// TIA Portal project "AutomationProjectLMF" (V16)

(* hardware
DEVICE "S7-1200 station_1"  S7-1200 Station
   slot 0: "Telaio di montaggio_0"  S7-1200 Rack  Rack  V1.0
   slot 1: "PLC_1"  CPU 1215C AC/DC/Rly  6ES7 215-1BG40-0XB0  V4.2
*)

// ===== PLC "PLC_1"  CPU 1215C AC/DC/Rly =====

VAR_GLOBAL   // PLC tag table "Tabella delle variabili standard"
   "ARM_UP" AT %Q0.5 : Bool;
   "ARM_DOWN" AT %Q0.4 : Bool;
   "ArmTopStop" AT %I0.4 : Bool;
   "ARM_FRONT" AT %Q0.2 : Bool;
   "ARM_BACK" AT %Q0.3 : Bool;
   "FullBackArm" AT %I0.2 : Bool;
   "ARM_CCLOCKWISE" AT %Q0.7 : Bool;
   "ARM_CLOCKWISE" AT %Q0.6 : Bool;
   "FullyClockwiseArm" AT %I0.5 : Bool;
   "GRIP_CLOSE" AT %Q0.1 : Bool;
   "GRIP_OPEN" AT %Q0.0 : Bool;
   "FullyOpenGripper" AT %I0.0 : Bool;
   "RotationalEncoder" AT %ID1000 : DInt;
   "RotationalCounter" AT %MW2 : UInt;
   "VerticalEncoder" AT %ID1004 : DInt;
   "VerticalCounter" AT %MW4 : UInt;
   "System_Byte" AT %MB1 : Byte;
   "FirstScan" AT %M1.0 : Bool;
   "DiagStatusUpdate" AT %M1.1 : Bool;
   "AlwaysTRUE" AT %M1.2 : Bool;
   "AlwaysFALSE" AT %M1.3 : Bool;
   "System_Byte(1)" AT %MB1 : Byte;
   "System_Byte(2)" AT %MB1 : Byte;
   "System_Byte(3)" AT %MB1 : Byte;
   "Clock_Byte" AT %MB0 : Byte;
   "Clock_10Hz" AT %M0.0 : Bool;
   "Clock_5Hz" AT %M0.1 : Bool;
   "Clock_2.5Hz" AT %M0.2 : Bool;
   "Clock_2Hz" AT %M0.3 : Bool;
   "Clock_1.25Hz" AT %M0.4 : Bool;
   "Clock_1Hz" AT %M0.5 : Bool;
   "Clock_0.625Hz" AT %M0.6 : Bool;
   "Clock_0.5Hz" AT %M0.7 : Bool;
   "ForceReset" AT %M7.0 : Bool;
   "ResetCompleted" AT %M7.1 : Bool;
   "FRONT_STOP" AT %M7.2 : Bool;
   "ArmHCounter" AT %I0.3 : Bool;
   "ObjectDetected" AT %I1.5 : Bool;
   "HTarget" AT %MB2 : Byte;
   "Stop" AT %M6.1 : Bool;
   "GripperCounter" AT %I0.1 : Bool;
   "Started" AT %M6.3 : Bool;
   "FirstTarget" AT %M6.4 : Bool;
   "SecondTarget" AT %M6.5 : Bool;
   "ThirdTarget" AT %M6.6 : Bool;
   "Reset" AT %M6.7 : Bool;
   "FourthTarget" AT %M7.3 : Bool;
   "FifthTarget" AT %M7.4 : Bool;
   "SixthTarget" AT %M7.5 : Bool;
   "Conveyor" AT %Q1.1 : Bool;
   "Cart_Command" AT %MB3 : Byte;
   "Receveid_values" AT %MB4 : Byte;
   "CartReady" AT %M8.0 : Bool;
END_VAR

DATA_BLOCK "TCP_msg"   // DB8
{ S7_Optimized_Access := 'TRUE' }
VERSION : 0.1
   VAR
      Send : Byte := 0;
      Receive : Byte;
   END_VAR
BEGIN
END_DATA_BLOCK

// folder: System blocks/Program resources

DATA_BLOCK "ArmHPulseCounter"   // DB1
{ S7_Optimized_Access := 'TRUE' }
AUTHOR : Simatic
FAMILY : IEC
NAME : CNTR
VERSION : 1.0
// stored: InstanceOfName IEC_COUNTER
"IEC_COUNTER"
BEGIN
END_DATA_BLOCK

DATA_BLOCK "GripperPulseCounter"   // DB2
{ S7_Optimized_Access := 'TRUE' }
AUTHOR : Simatic
FAMILY : IEC
NAME : CNTR
VERSION : 1.0
// stored: InstanceOfName IEC_COUNTER
"IEC_COUNTER"
BEGIN
END_DATA_BLOCK

DATA_BLOCK "PLC_1_Connection_DB"   // DB5
{ S7_Optimized_Access := 'TRUE' }
AUTHOR : SIMATIC
FAMILY : MC7Plus
NAME : TC_IP_v4
VERSION : 1.0
// stored: InstanceOfName TCON_IP_v4
"TCON_IP_v4"
BEGIN
   ID := 1;
   InterfaceId := 64;
   RemotePort := 2001;
   ActiveEstablished := true;
   RemoteAddress.ADDR[1] := 192;
   RemoteAddress.ADDR[2] := 168;
   RemoteAddress.ADDR[4] := 241;
END_DATA_BLOCK

// folder: (top level)

ORGANIZATION_BLOCK "Main"   // OB1, LAD, ProgramCycle
TITLE = "Main Program Sweep (Cycle)"
{ S7_Optimized_Access := 'TRUE' }
VERSION : 0.1
   VAR_INPUT
      Initial_Call : Bool;   // Initial call of this OB
      Remanence : Bool;   // =True, if remanent data are available
   END_VAR
   VAR_TEMP   // added for the SCL form of the ladder/FBD networks
      _w1 : Bool;
      _w2 : Bool;
      _w3 : Bool;
   END_VAR
BEGIN

REGION Network 1
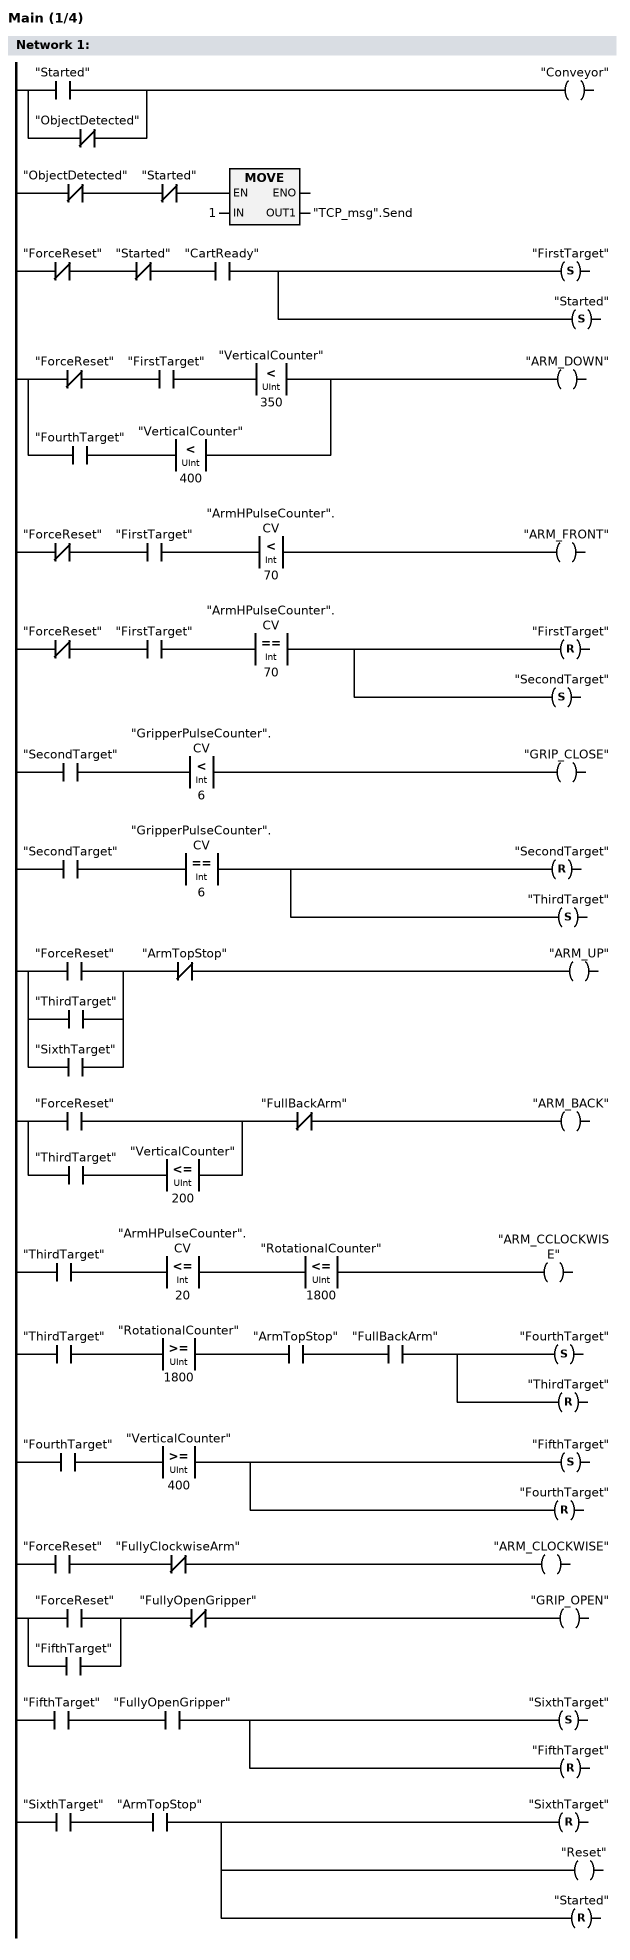
   RUNG wire#powerrail
      Contact( "Started" )
      wire#w1
      Coil( "Conveyor" )
   END_RUNG
   RUNG wire#powerrail
      I_Contact( "ObjectDetected" )
   END_RUNG wire#w1
   RUNG wire#powerrail
      I_Contact( "ObjectDetected" )
      I_Contact( "Started" )
      Move(in := 1, out1 => "TCP_msg".Send)
   END_RUNG
   RUNG wire#powerrail
      I_Contact( "ForceReset" )
      I_Contact( "Started" )
      Contact( "CartReady" )
      wire#w2
      S_Coil( "FirstTarget" )
   END_RUNG
   RUNG wire#w2
      S_Coil( "Started" )
   END_RUNG
   RUNG wire#powerrail
      I_Contact( "ForceReset" )
      Contact( "FirstTarget" )
      { S7_Templates := "SrcType := UInt" } LT_Contact(in1 := "VerticalCounter", in2 := 350)
      wire#w3
      Coil( "ARM_DOWN" )
   END_RUNG
   RUNG wire#powerrail
      Contact( "FourthTarget" )
      { S7_Templates := "SrcType := UInt" } LT_Contact(in1 := "VerticalCounter", in2 := 400)
   END_RUNG wire#w3
   RUNG wire#powerrail
      I_Contact( "ForceReset" )
      Contact( "FirstTarget" )
      { S7_Templates := "SrcType := Int" } LT_Contact(in1 := "ArmHPulseCounter".CV, in2 := 70)
      Coil( "ARM_FRONT" )
   END_RUNG
   RUNG wire#powerrail
      I_Contact( "ForceReset" )
      Contact( "FirstTarget" )
      { S7_Templates := "SrcType := Int" } EQ_Contact(in1 := "ArmHPulseCounter".CV, in2 := 70)
      wire#w4
      R_Coil( "FirstTarget" )
   END_RUNG
   RUNG wire#w4
      S_Coil( "SecondTarget" )
   END_RUNG
   RUNG wire#powerrail
      Contact( "SecondTarget" )
      { S7_Templates := "SrcType := Int" } LT_Contact(in1 := "GripperPulseCounter".CV, in2 := 6)
      Coil( "GRIP_CLOSE" )
   END_RUNG
   RUNG wire#powerrail
      Contact( "SecondTarget" )
      { S7_Templates := "SrcType := Int" } EQ_Contact(in1 := "GripperPulseCounter".CV, in2 := 6)
      wire#w5
      R_Coil( "SecondTarget" )
   END_RUNG
   RUNG wire#w5
      S_Coil( "ThirdTarget" )
   END_RUNG
   RUNG wire#powerrail
      Contact( "ForceReset" )
      wire#w6
      I_Contact( "ArmTopStop" )
      Coil( "ARM_UP" )
   END_RUNG
   RUNG wire#powerrail
      Contact( "ThirdTarget" )
   END_RUNG wire#w6
   RUNG wire#powerrail
      Contact( "SixthTarget" )
   END_RUNG wire#w6
   RUNG wire#powerrail
      Contact( "ForceReset" )
      wire#w7
      I_Contact( "FullBackArm" )
      Coil( "ARM_BACK" )
   END_RUNG
   RUNG wire#powerrail
      Contact( "ThirdTarget" )
      { S7_Templates := "SrcType := UInt" } LE_Contact(in1 := "VerticalCounter", in2 := 200)
   END_RUNG wire#w7
   RUNG wire#powerrail
      Contact( "ThirdTarget" )
      { S7_Templates := "SrcType := Int" } LE_Contact(in1 := "ArmHPulseCounter".CV, in2 := 20)
      { S7_Templates := "SrcType := UInt" } LE_Contact(in1 := "RotationalCounter", in2 := 1800)
      Coil( "ARM_CCLOCKWISE" )
   END_RUNG
   RUNG wire#powerrail
      Contact( "ThirdTarget" )
      { S7_Templates := "SrcType := UInt" } GE_Contact(in1 := "RotationalCounter", in2 := 1800)
      Contact( "ArmTopStop" )
      Contact( "FullBackArm" )
      wire#w8
      S_Coil( "FourthTarget" )
   END_RUNG
   RUNG wire#w8
      R_Coil( "ThirdTarget" )
   END_RUNG
   RUNG wire#powerrail
      Contact( "FourthTarget" )
      { S7_Templates := "SrcType := UInt" } GE_Contact(in1 := "VerticalCounter", in2 := 400)
      wire#w9
      S_Coil( "FifthTarget" )
   END_RUNG
   RUNG wire#w9
      R_Coil( "FourthTarget" )
   END_RUNG
   RUNG wire#powerrail
      Contact( "ForceReset" )
      I_Contact( "FullyClockwiseArm" )
      Coil( "ARM_CLOCKWISE" )
   END_RUNG
   RUNG wire#powerrail
      Contact( "ForceReset" )
      wire#w10
      I_Contact( "FullyOpenGripper" )
      Coil( "GRIP_OPEN" )
   END_RUNG
   RUNG wire#powerrail
      Contact( "FifthTarget" )
   END_RUNG wire#w10
   RUNG wire#powerrail
      Contact( "FifthTarget" )
      Contact( "FullyOpenGripper" )
      wire#w11
      S_Coil( "SixthTarget" )
   END_RUNG
   RUNG wire#w11
      R_Coil( "FifthTarget" )
   END_RUNG
   RUNG wire#powerrail
      Contact( "SixthTarget" )
      Contact( "ArmTopStop" )
      wire#w12
      R_Coil( "SixthTarget" )
   END_RUNG
   RUNG wire#w12
      Coil( "Reset" )
   END_RUNG
   RUNG wire#w12
      R_Coil( "Started" )
   END_RUNG
   // the same network as SCL:
   "Conveyor" := "Started" OR NOT "ObjectDetected";
   IF NOT "ObjectDetected" AND NOT "Started" THEN "TCP_msg".Send := 1; END_IF;
   IF NOT "ForceReset" AND NOT "Started" AND "CartReady" THEN
       "FirstTarget" := TRUE;
       "Started" := TRUE;
   END_IF;
   "ARM_DOWN" := (NOT "ForceReset" AND "FirstTarget" AND ("VerticalCounter" < 350)) OR ("FourthTarget" AND ("VerticalCounter" < 400));
   "ARM_FRONT" := NOT "ForceReset" AND "FirstTarget" AND ("ArmHPulseCounter".CV < 70);
   #_w1 := NOT "ForceReset" AND "FirstTarget" AND ("ArmHPulseCounter".CV = 70);
   IF #_w1 THEN
       "FirstTarget" := FALSE;
       "SecondTarget" := TRUE;
   END_IF;
   "GRIP_CLOSE" := "SecondTarget" AND ("GripperPulseCounter".CV < 6);
   #_w2 := "SecondTarget" AND ("GripperPulseCounter".CV = 6);
   IF #_w2 THEN
       "SecondTarget" := FALSE;
       "ThirdTarget" := TRUE;
   END_IF;
   "ARM_UP" := ("ForceReset" OR "ThirdTarget" OR "SixthTarget") AND NOT "ArmTopStop";
   "ARM_BACK" := ("ForceReset" OR ("ThirdTarget" AND ("VerticalCounter" <= 200))) AND NOT "FullBackArm";
   "ARM_CCLOCKWISE" := "ThirdTarget" AND ("ArmHPulseCounter".CV <= 20) AND ("RotationalCounter" <= 1800);
   IF "ThirdTarget" AND ("RotationalCounter" >= 1800) AND "ArmTopStop" AND "FullBackArm" THEN
       "FourthTarget" := TRUE;
       "ThirdTarget" := FALSE;
   END_IF;
   IF "FourthTarget" AND ("VerticalCounter" >= 400) THEN
       "FifthTarget" := TRUE;
       "FourthTarget" := FALSE;
   END_IF;
   "ARM_CLOCKWISE" := "ForceReset" AND NOT "FullyClockwiseArm";
   "GRIP_OPEN" := ("ForceReset" OR "FifthTarget") AND NOT "FullyOpenGripper";
   IF "FifthTarget" AND "FullyOpenGripper" THEN
       "SixthTarget" := TRUE;
       "FifthTarget" := FALSE;
   END_IF;
   #_w3 := "SixthTarget" AND "ArmTopStop";
   IF #_w3 THEN "SixthTarget" := FALSE; END_IF;
   "Reset" := #_w3;
   IF #_w3 THEN "Started" := FALSE; END_IF;
END_REGION

REGION Network 2: Reset
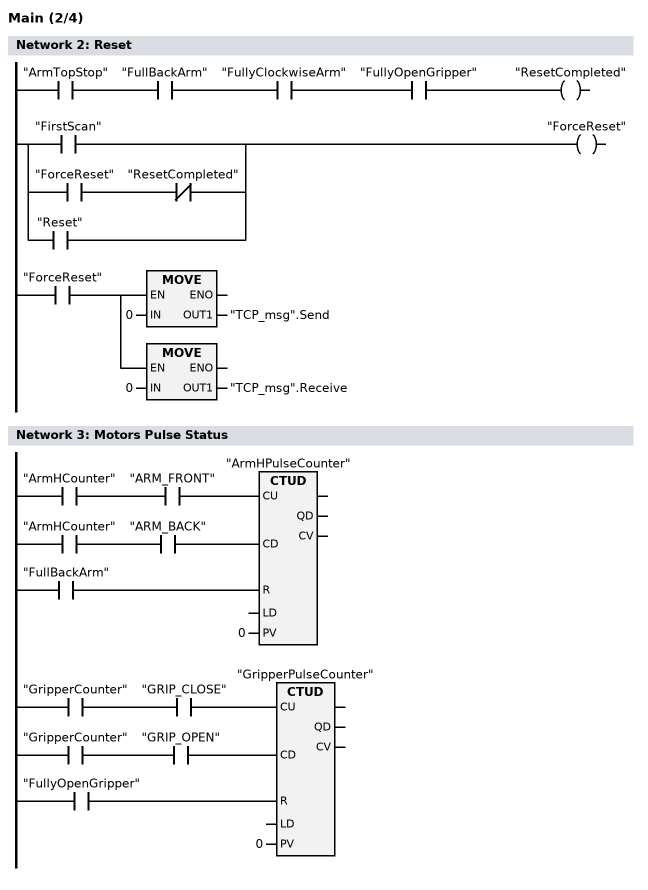
   RUNG wire#powerrail
      Contact( "ArmTopStop" )
      Contact( "FullBackArm" )
      Contact( "FullyClockwiseArm" )
      Contact( "FullyOpenGripper" )
      Coil( "ResetCompleted" )
   END_RUNG
   RUNG wire#powerrail
      Contact( "FirstScan" )
      wire#w1
      Coil( "ForceReset" )
   END_RUNG
   RUNG wire#powerrail
      Contact( "ForceReset" )
      I_Contact( "ResetCompleted" )
   END_RUNG wire#w1
   RUNG wire#powerrail
      Contact( "Reset" )
   END_RUNG wire#w1
   RUNG wire#powerrail
      Contact( "ForceReset" )
      wire#w2
      Move(in := 0, out1 => "TCP_msg".Send)
   END_RUNG
   RUNG wire#w2
      Move(in := 0, out1 => "TCP_msg".Receive)
   END_RUNG
   // the same network as SCL:
   "ResetCompleted" := "ArmTopStop" AND "FullBackArm" AND "FullyClockwiseArm" AND "FullyOpenGripper";
   "ForceReset" := "FirstScan" OR ("ForceReset" AND NOT "ResetCompleted") OR "Reset";
   IF "ForceReset" THEN
       "TCP_msg".Send := 0;
       "TCP_msg".Receive := 0;
   END_IF;
END_REGION

REGION Network 3: Motors Pulse Status
   "ArmHPulseCounter".CTUD(CU := "ArmHCounter" AND "ARM_FRONT",
                           CD := "ArmHCounter" AND "ARM_BACK",
                           R := "FullBackArm",
                           PV := 0);
   "GripperPulseCounter".CTUD(CU := "GripperCounter" AND "GRIP_CLOSE",
                           CD := "GripperCounter" AND "GRIP_OPEN",
                           R := "FullyOpenGripper",
                           PV := 0);
END_REGION

REGION Network 4: Encoder Status
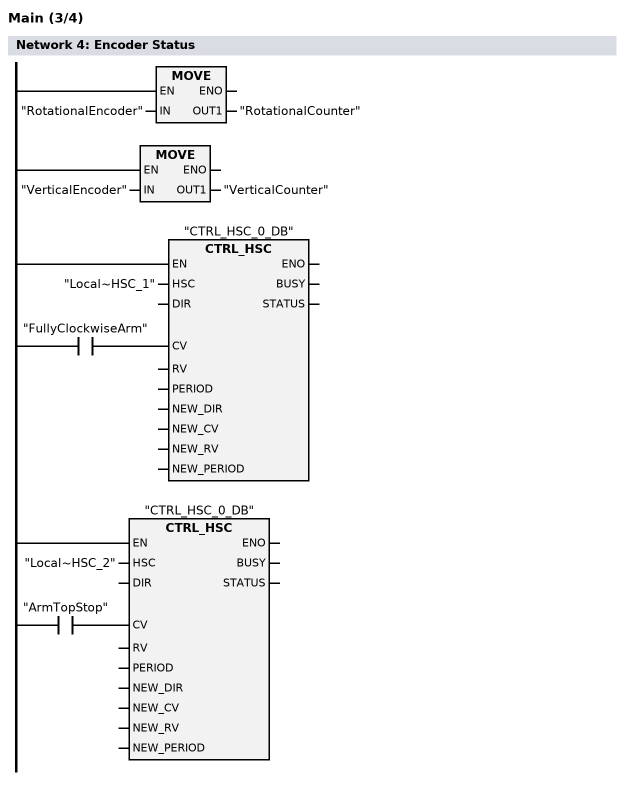
   "RotationalCounter" := "RotationalEncoder";
   "VerticalCounter" := "VerticalEncoder";
   "CTRL_HSC_0_DB"(HSC := "Local~HSC_1", CV := "FullyClockwiseArm");   // CTRL_HSC
   "CTRL_HSC_0_DB"(HSC := "Local~HSC_2", CV := "ArmTopStop");   // CTRL_HSC
END_REGION

REGION Network 5: Connection
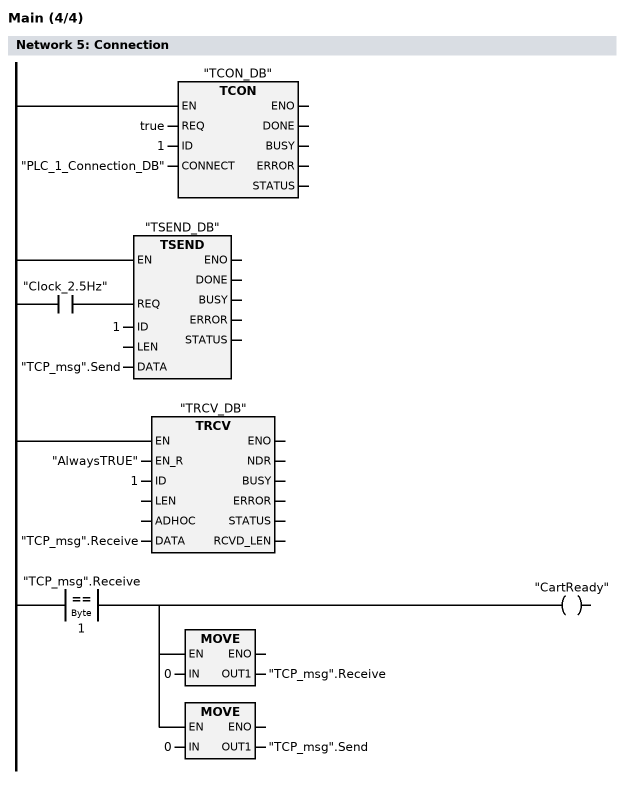
   "TCON_DB"(REQ := true, ID := 1, CONNECT := "PLC_1_Connection_DB");   // TCON
   "TSEND_DB"(REQ := "Clock_2.5Hz", ID := 1, DATA := "TCP_msg".Send);   // TSEND
   "TRCV_DB"(EN_R := "AlwaysTRUE", ID := 1, DATA := "TCP_msg".Receive);   // TRCV
   "CartReady" := "TCP_msg".Receive = 1;
   IF "CartReady" THEN
       "TCP_msg".Receive := 0;
       "TCP_msg".Send := 0;
   END_IF;
END_REGION
END_ORGANIZATION_BLOCK